ABB RAPID module: Module1.mod

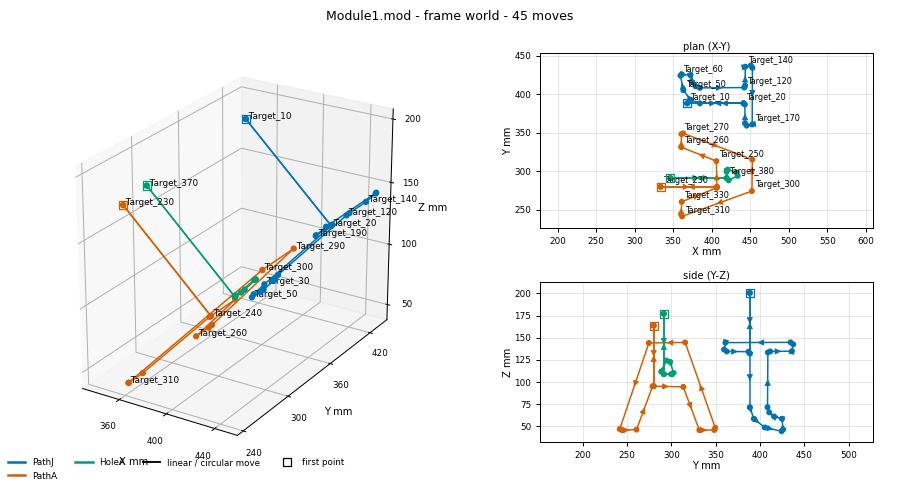
[picture p0: tool path of Module1.mod in frame world, 45 of 47 moves have a stored position in this frame; points joined in program order, loops and branches not executed]
MODULE Module1
        CONST robtarget Target_10:=[[96.084380669,84.821764131,-99.999819375],[0.707106377,0.000000835,-0.000000835,0.707107185],[0,0,0,0],[9E+09,9E+09,9E+09,9E+09,9E+09,9E+09]];
    CONST robtarget Target_20:=[[96.084380669,84.821528022,0.000180624],[0.707106377,0.000000835,-0.000000835,0.707107185],[0,-2,1,0],[9E+09,9E+09,9E+09,9E+09,9E+09,9E+09]];
    CONST robtarget Target_30:=[[96.084380669,167.821528022,0.000376594],[0.707106377,0.000000835,-0.000000835,0.707107185],[0,-2,1,0],[9E+09,9E+09,9E+09,9E+09,9E+09,9E+09]];
    CONST robtarget Target_40:=[[91.589002753,185.627739864,0.000418636],[0.707106377,0.000000835,-0.000000834,0.707107185],[0,-2,1,0],[9E+09,9E+09,9E+09,9E+09,9E+09,9E+09]];
    CONST robtarget Target_50:=[[79.180280025,199.166321883,0.000450602],[0.707106377,0.000000835,-0.000000835,0.707107185],[0,-2,1,0],[9E+09,9E+09,9E+09,9E+09,9E+09,9E+09]];
    CONST robtarget Target_60:=[[60.224636319,204.884514872,0.000464103],[0.707106377,0.000000835,-0.000000835,0.707107185],[0,-2,1,0],[9E+09,9E+09,9E+09,9E+09,9E+09,9E+09]];
    CONST robtarget Target_70:=[[58.571449711,202.20382584,0.000457774],[0.707106377,0.000000835,-0.000000835,0.707107185],[0,-2,1,0],[9E+09,9E+09,9E+09,9E+09,9E+09,9E+09]];
    CONST robtarget Target_80:=[[59.824807629,185.67479272,0.000418747],[0.707106377,0.000000835,-0.000000835,0.707107185],[0,-2,1,0],[9E+09,9E+09,9E+09,9E+09,9E+09,9E+09]];
    CONST robtarget Target_90:=[[68.767723776,182.060163698,0.000410213],[0.707106377,0.000000835,-0.000000835,0.707107185],[0,-2,1,0],[9E+09,9E+09,9E+09,9E+09,9E+09,9E+09]];
    CONST robtarget Target_100:=[[74.14818548,175.825780236,0.000395493],[0.707106377,0.000000835,-0.000000834,0.707107185],[0,-2,1,0],[9E+09,9E+09,9E+09,9E+09,9E+09,9E+09]];
    CONST robtarget Target_110:=[[76.084380669,167.821528022,0.000376594],[0.707106377,0.000000835,-0.000000835,0.707107185],[0,-2,1,0],[9E+09,9E+09,9E+09,9E+09,9E+09,9E+09]];
    CONST robtarget Target_120:=[[75.68245688,83.321528023,0.000177083],[0.707106377,0.000000834,-0.000000835,0.707107185],[0,-2,1,0],[9E+09,9E+09,9E+09,9E+09,9E+09,9E+09]];
    CONST robtarget Target_130:=[[73.084380669,81.821528022,0.000173541],[0.707106377,0.000000835,-0.000000835,0.707107185],[0,-2,1,0],[9E+09,9E+09,9E+09,9E+09,9E+09,9E+09]];
    CONST robtarget Target_140:=[[48.584380669,81.419604233,0.000172592],[0.707106377,0.000000834,-0.000000835,0.707107185],[0,-2,1,0],[9E+09,9E+09,9E+09,9E+09,9E+09,9E+09]];
    CONST robtarget Target_150:=[[47.084380669,70.821528022,0.000147569],[0.707106377,0.000000835,-0.000000835,0.707107185],[0,-1,1,0],[9E+09,9E+09,9E+09,9E+09,9E+09,9E+09]];
    CONST robtarget Target_160:=[[50.084380669,67.821528022,0.000140485],[0.707106377,0.000000835,-0.000000835,0.707107185],[0,-1,1,0],[9E+09,9E+09,9E+09,9E+09,9E+09,9E+09]];
    CONST robtarget Target_170:=[[123.584380669,68.223451811,0.000141434],[0.707106377,0.000000834,-0.000000835,0.707107185],[0,-2,1,0],[9E+09,9E+09,9E+09,9E+09,9E+09,9E+09]];
    CONST robtarget Target_180:=[[125.084380669,78.821528022,0.000166457],[0.707106377,0.000000835,-0.000000835,0.707107185],[0,-2,1,0],[9E+09,9E+09,9E+09,9E+09,9E+09,9E+09]];
    CONST robtarget Target_190:=[[122.084380669,81.821528022,0.000173541],[0.707106377,0.000000835,-0.000000835,0.707107185],[0,-2,1,0],[9E+09,9E+09,9E+09,9E+09,9E+09,9E+09]];
    CONST robtarget Target_200:=[[97.584380669,82.223451811,0.00017449],[0.707106377,0.000000835,-0.000000834,0.707107185],[0,-2,1,0],[9E+09,9E+09,9E+09,9E+09,9E+09,9E+09]];
    CONST robtarget Target_210:=[[96.084380669,84.821528022,0.000180624],[0.707106377,0.000000835,-0.000000835,0.707107185],[0,-2,1,0],[9E+09,9E+09,9E+09,9E+09,9E+09,9E+09]];
    CONST robtarget Target_220:=[[96.084380669,84.821764131,-99.999819375],[0.707106377,0.000000835,-0.000000835,0.707107185],[0,-1,1,0],[9E+09,9E+09,9E+09,9E+09,9E+09,9E+09]];
    CONST robtarget Target_230:=[[204.520079873,135.396087932,-99.999699965],[0.707106377,0.000000835,-0.000000835,0.707107185],[0,-2,1,0],[9E+09,9E+09,9E+09,9E+09,9E+09,9E+09]];
    CONST robtarget Target_240:=[[204.520079873,135.395851823,0.000300034],[0.707106377,0.000000835,-0.000000835,0.707107185],[0,-2,1,0],[9E+09,9E+09,9E+09,9E+09,9E+09,9E+09]];
    CONST robtarget Target_250:=[[171.109544621,136.494358922,0.000302627],[0.707106377,0.000000835,-0.000000835,0.707107185],[0,-2,1,0],[9E+09,9E+09,9E+09,9E+09,9E+09,9E+09]];
    CONST robtarget Target_260:=[[153.045748667,203.211008055,0.000460152],[0.707106377,0.000000834,-0.000000834,0.707107185],[0,-2,1,0],[9E+09,9E+09,9E+09,9E+09,9E+09,9E+09]];
    CONST robtarget Target_270:=[[136.239375779,202.966932031,0.000459576],[0.707106377,0.000000835,-0.000000835,0.707107185],[0,-2,1,0],[9E+09,9E+09,9E+09,9E+09,9E+09,9E+09]];
    CONST robtarget Target_280:=[[135.03489197,199.773741058,0.000452036],[0.707106377,0.000000835,-0.000000834,0.707107185],[0,-2,1,0],[9E+09,9E+09,9E+09,9E+09,9E+09,9E+09]];
    CONST robtarget Target_290:=[[169.035225221,67.946603757,0.000140781],[0.707106377,0.000000834,-0.000000834,0.707107185],[0,-2,1,0],[9E+09,9E+09,9E+09,9E+09,9E+09,9E+09]];
    CONST robtarget Target_300:=[[209.951577535,68.756612165,0.000142693],[0.707106377,0.000000835,-0.000000835,0.707107185],[0,-2,1,0],[9E+09,9E+09,9E+09,9E+09,9E+09,9E+09]];
    CONST robtarget Target_310:=[[242.811208671,201.558298439,0.000456249],[0.707106377,0.000000834,-0.000000835,0.707107185],[0,-2,2,0],[9E+09,9E+09,9E+09,9E+09,9E+09,9E+09]];
    CONST robtarget Target_320:=[[240.004260123,203.499506745,0.000460832],[0.707106377,0.000000835,-0.000000835,0.707107185],[0,-2,2,0],[9E+09,9E+09,9E+09,9E+09,9E+09,9E+09]];
    CONST robtarget Target_330:=[[223.867527121,202.400999647,0.000458239],[0.707106377,0.000000835,-0.000000835,0.707107185],[0,-2,2,0],[9E+09,9E+09,9E+09,9E+09,9E+09,9E+09]];
    CONST robtarget Target_340:=[[205.803731167,135.684350514,0.000300715],[0.707106377,0.000000834,-0.000000834,0.707107185],[0,-2,1,0],[9E+09,9E+09,9E+09,9E+09,9E+09,9E+09]];
    CONST robtarget Target_350:=[[204.520079873,135.395851823,0.000300034],[0.707106377,0.000000835,-0.000000835,0.707107185],[0,-2,1,0],[9E+09,9E+09,9E+09,9E+09,9E+09,9E+09]];
    CONST robtarget Target_360:=[[204.520079873,135.396087932,-99.999699965],[0.707106377,0.000000835,-0.000000835,0.707107185],[0,-2,1,0],[9E+09,9E+09,9E+09,9E+09,9E+09,9E+09]];
    CONST robtarget Target_370:=[[193.065343517,116.890641658,-99.999743659],[0.707106377,0.000000835,-0.000000835,0.707107185],[0,-2,1,0],[9E+09,9E+09,9E+09,9E+09,9E+09,9E+09]];
    CONST robtarget Target_380:=[[193.065343517,116.890405549,0.000256341],[0.707106377,0.000000835,-0.000000835,0.707107185],[0,-2,1,0],[9E+09,9E+09,9E+09,9E+09,9E+09,9E+09]];
    CONST robtarget Target_390:=[[195.963120996,113.113948414,0.000247424],[0.707106377,0.000000835,-0.000000834,0.707107185],[0,-2,1,0],[9E+09,9E+09,9E+09,9E+09,9E+09,9E+09]];
    CONST robtarget Target_400:=[[190.242874421,95.906185643,0.000206795],[0.707106377,0.000000835,-0.000000835,0.707107185],[0,-2,1,0],[9E+09,9E+09,9E+09,9E+09,9E+09,9E+09]];
    CONST robtarget Target_410:=[[186.077242157,97.848651869,0.000211382],[0.707106377,0.000000834,-0.000000835,0.707107185],[0,-2,1,0],[9E+09,9E+09,9E+09,9E+09,9E+09,9E+09]];
    CONST robtarget Target_420:=[[182.065617892,114.916465979,0.000251681],[0.707106377,0.000000835,-0.000000836,0.707107185],[0,-2,1,0],[9E+09,9E+09,9E+09,9E+09,9E+09,9E+09]];
    CONST robtarget Target_430:=[[184.884695755,116.890405549,0.000256341],[0.707106377,0.000000835,-0.000000835,0.707107185],[0,-2,1,0],[9E+09,9E+09,9E+09,9E+09,9E+09,9E+09]];
    CONST robtarget Target_440:=[[193.065343517,116.890405549,0.000256341],[0.707106377,0.000000835,-0.000000835,0.707107185],[0,-2,1,0],[9E+09,9E+09,9E+09,9E+09,9E+09,9E+09]];
    CONST robtarget Target_450:=[[193.065343517,116.890641658,-99.999743659],[0.707106377,0.000000835,-0.000000835,0.707107185],[0,-2,1,0],[9E+09,9E+09,9E+09,9E+09,9E+09,9E+09]];
    CONST jointtarget Home:=[[0,0,0,0,0,0],[9E+09,9E+09,9E+09,9E+09,9E+09,9E+09]];
    CONST jointtarget Mid:=[[82.602612887,7.641917879,33.301307391,-53.615287683,44.510328941,0.000000101],[9E+09,9E+09,9E+09,9E+09,9E+09,9E+09]];
!***********************************************************
    !
    ! Module:  Module1
    !
    ! Description:
    !   <Insert description here>
    !
    ! Author: allan
    !
    ! Version: 1.0
    !
    !***********************************************************


    !***********************************************************
    !
    ! Procedure main
    !
    !   This is the entry point of your program
    !
    !***********************************************************
    PROC main()
        Homing;
        Midpoint;
        PathJ;
        PathA;
        HoleA;
        Midpoint;
        Homing;

    ENDPROC
    PROC PathJ()
        MoveL Target_10,v100,z10,Marcador3\WObj:=tablero3;
        MoveL Target_20,v100,z10,Marcador3\WObj:=tablero3;
        MoveL Target_30,v100,z10,Marcador3\WObj:=tablero3;
        MoveL Target_40,v100,z10,Marcador3\WObj:=tablero3;
        MoveL Target_50,v100,z10,Marcador3\WObj:=tablero3;
        MoveL Target_60,v100,z10,Marcador3\WObj:=tablero3;
        MoveL Target_70,v100,z10,Marcador3\WObj:=tablero3;
        MoveL Target_80,v100,z10,Marcador3\WObj:=tablero3;
        MoveL Target_90,v100,z10,Marcador3\WObj:=tablero3;
        MoveL Target_100,v100,z10,Marcador3\WObj:=tablero3;
        MoveL Target_110,v100,z10,Marcador3\WObj:=tablero3;
        MoveL Target_120,v100,z10,Marcador3\WObj:=tablero3;
        MoveL Target_130,v100,z10,Marcador3\WObj:=tablero3;
        MoveL Target_140,v100,z10,Marcador3\WObj:=tablero3;
        MoveL Target_150,v100,z10,Marcador3\WObj:=tablero3;
        MoveL Target_160,v100,z10,Marcador3\WObj:=tablero3;
        MoveL Target_170,v100,z10,Marcador3\WObj:=tablero3;
        MoveL Target_180,v100,z10,Marcador3\WObj:=tablero3;
        MoveL Target_190,v100,z10,Marcador3\WObj:=tablero3;
        MoveL Target_200,v100,z10,Marcador3\WObj:=tablero3;
        MoveL Target_210,v100,z10,Marcador3\WObj:=tablero3;
        MoveL Target_220,v100,z10,Marcador3\WObj:=tablero3;
    ENDPROC
    PROC PathA()
        MoveL Target_230,v80,z5,Marcador3\WObj:=tablero3;
        MoveL Target_240,v80,z5,Marcador3\WObj:=tablero3;
        MoveL Target_250,v80,z5,Marcador3\WObj:=tablero3;
        MoveL Target_260,v80,z5,Marcador3\WObj:=tablero3;
        MoveL Target_270,v80,z5,Marcador3\WObj:=tablero3;
        MoveL Target_280,v80,z5,Marcador3\WObj:=tablero3;
        MoveL Target_290,v80,z5,Marcador3\WObj:=tablero3;
        MoveL Target_300,v80,z5,Marcador3\WObj:=tablero3;
        MoveL Target_310,v80,z5,Marcador3\WObj:=tablero3;
        MoveL Target_320,v80,z5,Marcador3\WObj:=tablero3;
        MoveL Target_330,v80,z5,Marcador3\WObj:=tablero3;
        MoveL Target_340,v80,z5,Marcador3\WObj:=tablero3;
        MoveL Target_350,v80,z5,Marcador3\WObj:=tablero3;
        MoveL Target_360,v80,z5,Marcador3\WObj:=tablero3;
    ENDPROC
    PROC HoleA()
        MoveL Target_370,v100,z10,Marcador3\WObj:=tablero3;
        MoveL Target_380,v100,z10,Marcador3\WObj:=tablero3;
        MoveL Target_390,v100,z10,Marcador3\WObj:=tablero3;
        MoveL Target_400,v100,z10,Marcador3\WObj:=tablero3;
        MoveL Target_410,v100,z10,Marcador3\WObj:=tablero3;
        MoveL Target_420,v100,z10,Marcador3\WObj:=tablero3;
        MoveL Target_430,v100,z10,Marcador3\WObj:=tablero3;
        MoveL Target_440,v100,z10,Marcador3\WObj:=tablero3;
        MoveL Target_450,v100,z10,Marcador3\WObj:=tablero3;
    ENDPROC
    PROC Homing()
        MoveAbsJ Home,v100,z10,Marcador3\WObj:=tablero3;
    ENDPROC
    PROC Midpoint()
        MoveAbsJ Mid,v100,z5,Marcador3\WObj:=tablero3;
    ENDPROC
ENDMODULE
